% RSLogix 500 project PROJECT 1  CGT PART Challenge.RSS, saved by version 8.30.00.16 %
PROJECT "UNTITLED"    % processor: Bul.1763 MicroLogix 1100 Series B %

PROGRAM FILES
  LAD 2 "SECTIONS"  4 rungs
  LAD 3 "INPUTS"  4 rungs
  LAD 4 "LOGIC"  1 rungs
  LAD 5 "OUTPUT"  3 rungs

DATA FILES
  O0 OUTPUT  4 elements
  I1 INPUT  6 elements
  S2 STATUS  66 elements
  B3 BINARY  1 elements
  T4 TIMER  1 elements
  C5 COUNTER  1 elements
  R6 CONTROL  1 elements
  N7 INTEGER  1 elements
  F8 FLOAT  1 elements

LADDER 2 "SECTIONS"
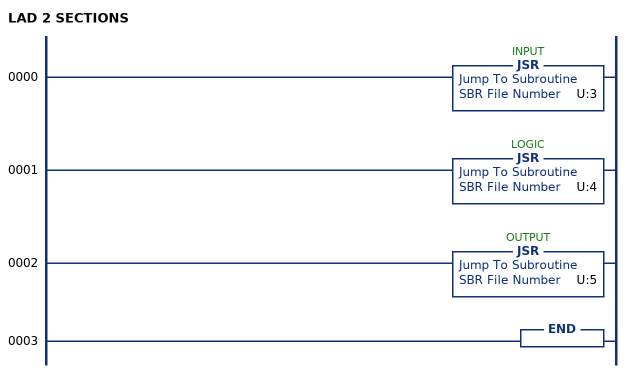
% Rung: 0 %  % edit flag set %
SOR JSR U:3 EOR
%   U:3  "INPUT" %
% Rung: 1 %  % edit flag set %
SOR JSR U:4 EOR
%   U:4  "LOGIC" %
% Rung: 2 %  % edit flag set %
SOR JSR U:5 EOR
%   U:5  "OUTPUT" %
% Rung: 3 %
SOR END EOR

LADDER 3 "INPUTS"
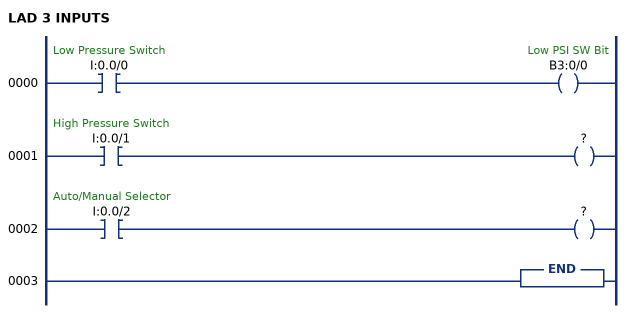
% Rung: 0 %  % edit flag set %
SOR XIC I:0.0/0 OTE B3:0/0 EOR
%   I:0.0/0  "Low Pressure Switch" %
%   B3:0/0  "Low PSI SW Bit" %
% Rung: 1 %  % edit flag set %
SOR XIC I:0.0/1 OTE ? EOR
%   I:0.0/1  "High Pressure Switch" %
% Rung: 2 %  % edit flag set %
SOR XIC I:0.0/2 OTE ? EOR
%   I:0.0/2  "Auto/Manual Selector" %
% Rung: 3 %  % edit flag set %
SOR END EOR

LADDER 5 "OUTPUT"
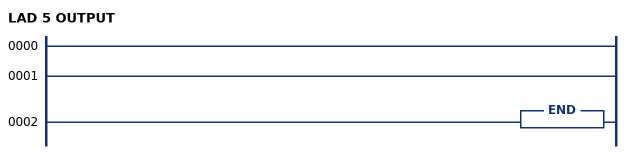
% Rung: 0 %  % edit flag set %
SOR EOR
% Rung: 1 %  % edit flag set %
SOR EOR
% Rung: 2 %  % edit flag set %
SOR END EOR
